PROGRAM MAIN
VAR
	myTimer					: TON;
	randomNumberGenerator	: DRAND();
	randomNumber			: LREAL;
	count					: WORD;
END_VAR

(*
	■ What is exchanged between Twincat Plc and Deskval Workbench ?  							
						Deskval Workbech exchanges its built-in AdsTags in a directional manner. 
						Deskval Workbench exchanges its built-in BatchTags, in a Readonly manner.	
	■ What is required in the Plc project ?
			Twincat Plc Project should have a Global Variable List, named as Deskval with a specific content. It is provided in this project.
					
						
	■ AdsTags				┌───────────────────────────────────────────────────────────────┐		┌───────────────────────────┐
							│ 						Twincat Plc Project         			│		│ 	  Deskval Workbench 	│    
							├───────────────────────────────────────────────────────────────┤		├───────────────────────────┤
							│															 	│		│         Ads Tags   		│     
							│															 	│		│							│                    
			┌────────────── │ 	AdsTagsFromDeskval_Boolean		AdsTagsToDeskval_Boolean	│ ────	► 128 Boolean	128 Boolean ►  ──────────────┐
			│	┌────────── │ 	AdsTagsFromDeskval_Double		AdsTagsToDeskval_Double		│ ────	► 64 Double		64 Double  	►  ──────────┐	 │
			│	│	┌──────	│ 	AdsTagsFromDeskval_String		AdsTagsToDeskval_String		│ ────	► 32 String    	32 String	►  ──────┐	 │	 │
			│	│	│		└───────────────────────────────────────────────────────────────┘		└───────────────────────────┘		 │	 │	 │
			│	│	└────────────────────────────────────────────────────────────────────────────────────────────────────────────────────┘	 │	 │
			│	└────────────────────────────────────────────────────────────────────────────────────────────────────────────────────────────┘	 │
			└────────────────────────────────────────────────────────────────────────────────────────────────────────────────────────────────────┘	

	■ BatchTags				┌───────────────────────────────────────────────────────────────┐		┌───────────────────────────┐
							│ 						Twincat Plc Project         			│		│ 	  Deskval Workbench* 	│    
							├───────────────────────────────────────────────────────────────┤		├───────────────────────────┤
							│															 	│		│       Batch Tags  		│     
							│							BatchTags							│ ◄───►	│		 32 String			│    
							└───────────────────────────────────────────────────────────────┘		└───────────────────────────┘			
			¹ If a Deskval BatchTag is configured to get its value from Ads, then Deskval will Read it from the Plc

	────────────────────────────────────────────────────────────────────────────────────────────────────
	Description : This is a Sample Plc Program to demonstrate Ads Communication with Deskval Workbench.
	──────────────────────────────────────────────────────────────────────────────────────────────────── *)
myTimer(IN:=TRUE, PT:=T#1S);

// On Timer Tick
IF(myTimer.Q) THEN
	
	//Get a Random Number
	randomNumberGenerator(Seed:=17, Num=>randomNumber);		
	
	// Write to First Boolean Tag
	Deskval.AdsTagsToDeskval_Boolean[0] := NOT(Deskval.AdsTagsToDeskval_Boolean[0]);
	
	// Write to Second Num Tag
	Deskval.AdsTagsToDeskval_Double[1] 	:= randomNumber*100;
	
	// Write to Third String Tag
	Deskval.AdsTagsToDeskval_String[2] 	:= CONCAT('Count ',WORD_TO_STRING(count));
	
	// Write To Fourth Batch Tag
	Deskval.BatchTags[3] 				:= CONCAT('Some Batch ',WORD_TO_STRING(count));
	
	// Reset Timer
	myTimer(IN:=FALSE);

	//Increment count
	count := count + 1;
END_IF

END_PROGRAM

(* stored: Version 1.1.0.1, ProductVersion 3.1.4024.12
   POU MAIN: Id {b0d9c06b-cc2b-4257-a6db-fed8bdb41f30}, SpecialFunc None *)
